// TIA Portal V18 export
FUNCTION_BLOCK "Frequency_Trans"   // FB3, LAD
{ S7_Optimized_Access := 'FALSE' }
// stored: SetENOAutomatically false
   VAR_INPUT
      I_Frequency : Real;
   END_VAR
   VAR_OUTPUT
      Q_Frequency { ExternalAccessible := 'False'; ExternalVisible := 'False'; ExternalWritable := 'False'} : Word;
      Q_Frequency_Trans : Array[0..1] of Byte;
   END_VAR
   VAR_IN_OUT
      IO_Frequency_Status { ExternalAccessible := 'False'; ExternalVisible := 'False'; ExternalWritable := 'False'} : Int;
   END_VAR
   VAR_TEMP
      T_Frequency_Tmp1 : Real;
      T_Frequency_Tmp2 : Byte;
   END_VAR
BEGIN

REGION Network 1 (SCL): Frequency Calc
   #T_Frequency_Tmp1 := "LGF_ScaleLinear"(x := #I_Frequency,
                                          x1 := 0.0,
                                          y1 := 49152.0,
                                          x2 := 100.0,
                                          y2 := 65535.0,
                                          yMin := 49152.0,
                                          yMax := 65535.0,
                                          error => "System_Error".System_Error[1].%X3,
                                          status => #IO_Frequency_Status);
   #Q_Frequency := ROUND(#T_Frequency_Tmp1);
   #T_Frequency_Tmp2 := #Q_Frequency_Trans[0];
   #Q_Frequency_Trans[0] := #Q_Frequency_Trans[1];
   #Q_Frequency_Trans[1] := #T_Frequency_Tmp2;
END_REGION
END_FUNCTION_BLOCK
